{attribute 'qualified_only'}
{attribute 'strict'}
TYPE E_MMStationBuffer :
(
	eMMStationBuffer_PreProcess		:= 0,
	eMMStationBuffer_PostProcess	:= 1
);
END_TYPE

(* stored: Version 1.1.0.1, ProductVersion 3.1.4024.5
   EnumerationTextList E_MMStationBuffer: Id {65f31e5a-b1b5-44e1-bb3d-a745088acb42} *)
